{attribute addProperty BoxType "KL8001"}
{attribute addProperty Id "State_0AT %I*USINT000Data_In_0AT %I*UINT000State_1AT %I*USINT000Data_In_1AT %I*UINT000State_2AT %I*USINT000Data_In_2AT %I*UINT000State_ExtAT %I*USINT000Ctrl_0AT %Q*USINT000Data_Out_0AT %Q*UINT000Ctrl_1AT %Q*USINT000Data_Out_1AT %Q*UINT000Ctrl_2AT %Q*USINT000Data_Out_2AT %Q*UINT000Ctrl_ExtAT %Q*USINT000"}
{attribute addProperty CRC "1692418787"}
{attribute addProperty SizeInBites "0"}
{attribute addProperty SizeInBytes "0"}
TYPE Channel_64E042E3 :
STRUCT
	{attribute addProperty Name "State_0"}
	State_0 AT %I* : USINT;
	{attribute addProperty Name "Data_In_0"}
	Data_In_0 AT %I* : UINT;
	{attribute addProperty Name "State_1"}
	State_1 AT %I* : USINT;
	{attribute addProperty Name "Data_In_1"}
	Data_In_1 AT %I* : UINT;
	{attribute addProperty Name "State_2"}
	State_2 AT %I* : USINT;
	{attribute addProperty Name "Data_In_2"}
	Data_In_2 AT %I* : UINT;
	{attribute addProperty Name "State_Ext"}
	State_Ext AT %I* : USINT;
	{attribute addProperty Name "Ctrl_0"}
	Ctrl_0 AT %Q* : USINT;
	{attribute addProperty Name "Data_Out_0"}
	Data_Out_0 AT %Q* : UINT;
	{attribute addProperty Name "Ctrl_1"}
	Ctrl_1 AT %Q* : USINT;
	{attribute addProperty Name "Data_Out_1"}
	Data_Out_1 AT %Q* : UINT;
	{attribute addProperty Name "Ctrl_2"}
	Ctrl_2 AT %Q* : USINT;
	{attribute addProperty Name "Data_Out_2"}
	Data_Out_2 AT %Q* : UINT;
	{attribute addProperty Name "Ctrl_Ext"}
	Ctrl_Ext AT %Q* : USINT;
END_STRUCT
END_TYPE

(* stored: Version 1.2.0.0, ProductVersion 3.1.4024.9
   DUT Channel_64E042E3: Id {3e5f7e2d-fba5-4b08-821b-5c8ab2db695e} *)
